FUNCTION F_UpdateValue
VAR_INPUT
	stValueStructure : REFERENCE TO ST_SampleValue;
END_VAR
VAR
END_VAR

stValueStructure.nNumber := stValueStructure.nNumber + 1;

END_FUNCTION

(* stored: Version 1.1.0.1, ProductVersion 3.1.4024.16
   POU F_UpdateValue: Id {4aa8a255-252e-4f00-bdc3-1baf10f181a3}, SpecialFunc None *)
